% RSLogix 500 project ROTAMETER_BAK011.RSS, saved by version 8.30.00.16 %
PROJECT "UNTITLED"    % processor: Bul.1763 MicroLogix 1100 Series B %

PROGRAM FILES
  LAD 2 "MAIN"  2 rungs
  LAD 3 "CONTROLS"  8 rungs

DATA FILES
  O0 OUTPUT  4 elements
  I1 INPUT  6 elements
  S2 STATUS  66 elements
  B3 BINARY  2 elements
  T4 TIMER  2 elements
  C5 COUNTER  1 elements
  R6 CONTROL  1 elements
  N7 INTEGER  1 elements
  F8 FLOAT  4 elements

LADDER 2 "MAIN"
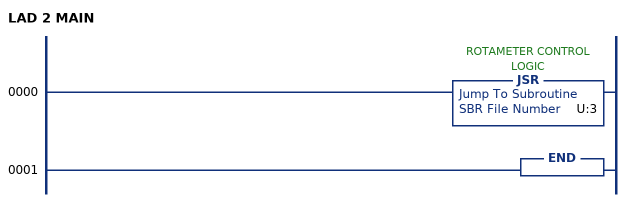
% Rung: 0 %
SOR JSR U:3 EOR
%   U:3  "ROTAMETER CONTROL LOGIC" %
% Rung: 1 %
SOR END EOR

LADDER 3 "CONTROLS"
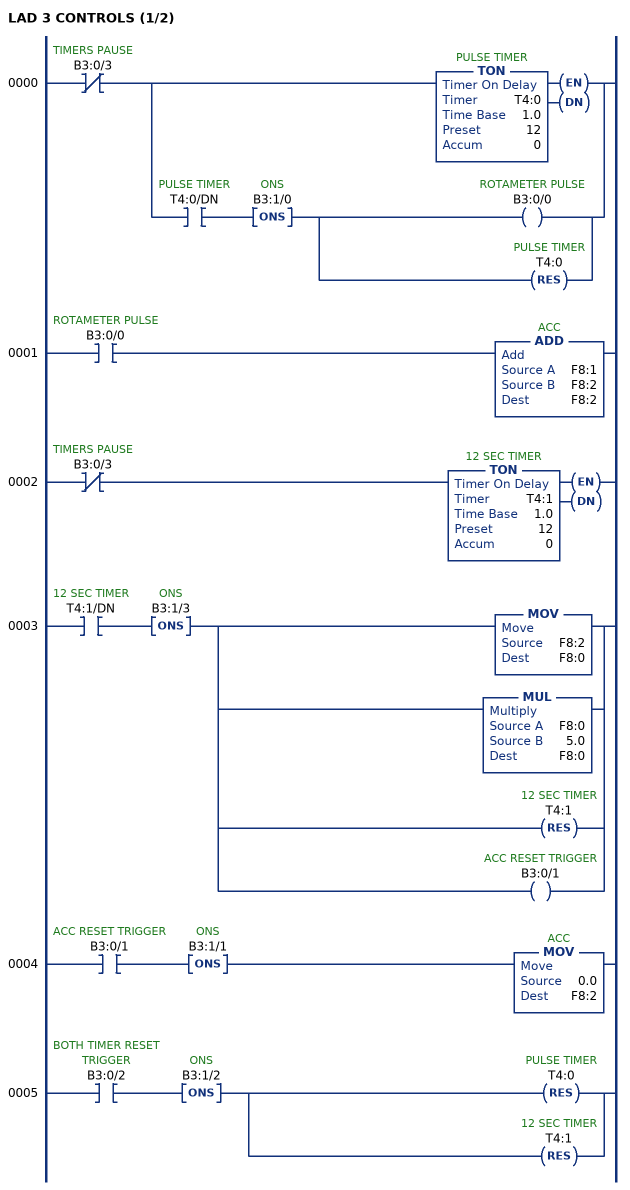
% Rung: 0 %
SOR XIO B3:0/3 BST TON T4:0 1.0 12 0 NXB XIC T4:0/DN ONS B3:1/0 BST OTE B3:0/0 NXB RES T4:0 BND BND EOR
%   B3:0/3  "TIMERS PAUSE" %
%   T4:0  "PULSE TIMER" %
%   B3:1/0  "ONS" %
%   B3:0/0  "ROTAMETER PULSE" %
% Rung: 1 %
SOR XIC B3:0/0 ADD F8:1 F8:2 F8:2 EOR
%   B3:0/0  "ROTAMETER PULSE" %
%   F8:1  "ROTEAMETER K-FACTOR" %
%   F8:2  "ACC" %
% Rung: 2 %
SOR XIO B3:0/3 TON T4:1 1.0 12 0 EOR
%   B3:0/3  "TIMERS PAUSE" %
%   T4:1  "12 SEC TIMER" %
% Rung: 3 %
SOR XIC T4:1/DN ONS B3:1/3 BST MOV F8:2 F8:0 NXB MUL F8:0 5.0 F8:0 NXB RES T4:1 NXB OTE B3:0/1 BND EOR
%   T4:1  "12 SEC TIMER" %
%   B3:1/3  "ONS" %
%   F8:2  "ACC" %
%   B3:0/1  "ACC RESET TRIGGER" %
% Rung: 4 %
SOR XIC B3:0/1 ONS B3:1/1 MOV 0.0 F8:2 EOR
%   B3:0/1  "ACC RESET TRIGGER" %
%   B3:1/1  "ONS" %
%   F8:2  "ACC" %
% Rung: 5 %
SOR XIC B3:0/2 ONS B3:1/2 BST RES T4:0 NXB RES T4:1 BND EOR
%   B3:0/2  "BOTH TIMER RESET TRIGGER" %
%   B3:1/2  "ONS" %
%   T4:0  "PULSE TIMER" %
%   T4:1  "12 SEC TIMER" %

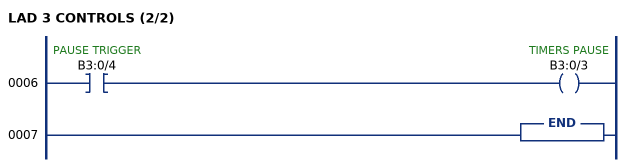
% Rung: 6 %
SOR XIC B3:0/4 OTE B3:0/3 EOR
%   B3:0/4  "PAUSE TRIGGER" %
%   B3:0/3  "TIMERS PAUSE" %
% Rung: 7 %
SOR END EOR

DATA TABLE (non-zero values as saved)
DATA T4
% .PRE .ACC %
% T4:0 % 12 0
% T4:1 % 12 0
DATA F8
% F8:0 % 0 6.3 0 0
